FUNCTION_BLOCK Track EXTENDS Objective IMPLEMENTS iTrack
VAR_INPUT
END_VAR
VAR_OUTPUT
END_VAR
VAR
	{attribute 'hide'}
	internalOTCID			: OTCID;	// internal track id for use with MC_ActivateTrack
	internalId				: INT;	// numeric track desigination i.e. "Track 1"
	internalMoverList : MoverList;	// working list of movers on this track
	internalIdIsSet			: BOOL; // track ID has been set, it is now ok to find the track OTCID
	internalOTCIDIsSet		: BOOL;	// track OTCID has been set, track commands can now be run
	internalLength			: LREAL; // length of track
END_VAR

PROPERTY CurrentMoverCount : DINT
GET
CurrentMoverCount := RegisteredMoverCount;
END_GET
END_PROPERTY

PROPERTY CurrentMoverList : iMoverList
GET
CurrentMoverList := internalMoverList;
END_GET
END_PROPERTY

METHOD Cyclic : BOOL
VAR
	nXpuTracks : UINT;
END_VAR
VAR_INST
	nState : TrackCyclicState;
END_VAR
IF internalIdIsSet AND NOT internalOTCIDIsSet THEN
	CASE nState OF
		TrackCyclicState.WAIT_FOR_ENV:	// wait for environment
			IF Mediator.EnvironmentIsReady THEN
				nState := TrackCyclicState.CHECK_ZERO_CASE;
			END_IF
		
		TrackCyclicState.CHECK_ZERO_CASE: // check for zero special case
			IF (internalId = 0) THEN
				// zero does not require initialization
				nState := TrackCyclicState.SET_INITIALIZED;
			ELSE
				nState := TrackCyclicState.CHECK_TRACK_COUNT;
			END_IF;
	
		TrackCyclicState.CHECK_TRACK_COUNT:	// check for track count
			nXpuTracks := Mediator.XPU.P_TrackCount;
			IF (internalId > UINT_TO_INT(nXpuTracks)) THEN
				// more tracks declared than defined in the XPU
				// this is considered deilberate and OK, no further initialization required
				nState := TrackCyclicState.SET_INITIALIZED;
			ELSE
				nState := TrackCyclicState.GET_OTCID;
			END_IF;
				
		TrackCyclicState.GET_OTCID: // get otcid
			internalOTCID := Mediator.XPU.P_TrackOids[internalId];
			nState :=TrackCyclicState.GET_LENGTH;
			
		TrackCyclicState.GET_LENGTH: // get length of track
			internalLength := Mediator.XPU.TrackTcIo(INT_TO_UINT(internalId)).GetLength();
			nState :=TrackCyclicState.SET_INITIALIZED;
			
		TrackCyclicState.SET_INITIALIZED: // set intitialized and rewind
			nState := TrackCyclicState.WAIT_FOR_ENV;
			internalOTCIDIsSet := TRUE;
			
	END_CASE
END_IF
END_METHOD

PROPERTY Id : INT
GET
Id := internalId;
END_GET
SET
internalId := Id;
// internal flag noting this value has been set this allows 0 (special case) to be used
internalIdIsSet := TRUE;
END_SET
END_PROPERTY

PROPERTY isInitialized : bool
GET
isInitialized := internalIdIsSet and internalOTCIDIsSet;
END_GET
END_PROPERTY

PROPERTY Length : LREAL
GET
END_GET
SET
Length := internalLength;
END_SET
END_PROPERTY

PROPERTY OTCID : OTCID
GET
OTCID := internalOTCID;
END_GET
SET
internalOTCID := OTCID;
// internal flag, pauses track methods until fbxtsenvironment has provided OTCIDs for each track
internalOTCIDIsSet := TRUE;
END_SET
END_PROPERTY

METHOD RegisterMover : BOOL
VAR_INPUT
    NewMover : REFERENCE TO Mover;
END_VAR
VAR
	i : ULINT;
END_VAR
// call the parent function
SUPER^.RegisterMover(NewMover);

// update the internal MoverList
// this saves us the time of generating it on every call to CurrentMoverCount
internalMoverList.UnregisterAll();

FOR i := 1 TO SIZEOF(internalRegisteredMovers) / SIZEOF(internalRegisteredMovers[1]) DO
    IF internalRegisteredMovers[i] <> 0 THEN
		internalMoverList.RegisterMover(internalRegisteredMovers[i]^);
	END_IF
END_FOR;
END_METHOD

METHOD UnregisterAll : BOOL
VAR_INPUT
END_VAR
// call the parent function
SUPER^.UnregisterAll();

// update the internal MoverList
// this saves us the time of generating it on every call to CurrentMoverCount
internalMoverList.UnregisterAll();
END_METHOD

METHOD UnregisterMover : BOOL
VAR_INPUT
    RemovingMover : REFERENCE TO Mover;
END_VAR
VAR
	i : ULINT;
END_VAR
// call the parent function
SUPER^.UnregisterMover(RemovingMover);

// update the internal MoverList
// this saves us the time of generating it on every call to CurrentMoverCount
internalMoverList.UnregisterAll();

FOR i := 0 TO SIZEOF(RegisteredMovers) / SIZEOF(internalRegisteredMovers[1]) - 1 DO
    IF internalRegisteredMovers[i] <> 0 THEN
		internalMoverList.RegisterMover(internalRegisteredMovers[i]^);
	END_IF
END_FOR;
END_METHOD

END_FUNCTION_BLOCK

(* stored: Version 1.1.0.1, ProductVersion 3.1.4026.8
   POU Track: Id {1d568bee-17b0-45d9-8c81-c6842c2a11d5}, SpecialFunc None
   Folder Methods: Id {39635f7a-3c34-4d67-b666-c6e08a70323b}
   Folder Properties: Id {5266f954-d54f-4746-897a-a6f4b18b8998}
   Property CurrentMoverCount: Id {2d1d239b-a67a-0e41-2ac7-acd8761cf4c8}
   Get Get: Id {c0df9483-acae-0f74-08b2-039449688a39}
   Property CurrentMoverList: Id {359f7362-4b29-0531-16e4-30c0573c9a91}
   Get Get: Id {60bc68b5-e5db-0d98-23eb-ecfa5a77a233}
   Method Cyclic: Id {0fbacee0-46ef-088c-34f0-d7cb5b41b934}
   Property Id: Id {bc141487-48e4-021d-1b8b-19fa2c77c46e}
   Get Get: Id {5dbdca49-4776-084f-23a4-b7b52bdccbfc}
   Set Set: Id {8e0384d9-fde2-0570-1441-0e0a49713398}
   Property isInitialized: Id {a010b7aa-b890-0ceb-3883-720b25186af2}
   Get Get: Id {8d3e9ef0-8df9-0a5c-34fa-bc058f56c77c}
   Property Length: Id {40cd32c0-bcdb-090a-2c41-7be7aeca95b1}
   Get Get: Id {12c0b740-e474-0caa-3d9f-c9c82397dae1}
   Set Set: Id {c74af95d-1365-01dd-05a7-8fb2224ded8b}
   Property OTCID: Id {dcb2dd98-b4d1-0928-1caf-998c96e183e9}
   Get Get: Id {2c637409-cdfd-0044-03ac-42f38e6d51b4}
   Set Set: Id {0ae5c3d3-9ea8-01d6-15e0-675b4a5b4cb0}
   Method RegisterMover: Id {91ee63c8-16e6-0d11-1bc4-051a0b49e848}
   Method UnregisterAll: Id {331df7c2-5517-0c9f-2789-611ea232bb66}
   Method UnregisterMover: Id {81fa567d-a876-0c41-1aea-870e51858476} *)
